FUNCTION alg_a_gripperclose : BOOL
VAR_INPUT
	state: STATE;
END_VAR

alg_a_gripperclose := state.dvar_M_example_controller_a_gripperclose;

END_FUNCTION

(* stored: Version 1.1.0.1, ProductVersion 3.1.4022.18
   POU alg_a_gripperclose: Id {d84ed6f0-d8d8-4aed-84c4-679a72b972a7}, SpecialFunc None *)
